// TwinCAT 3 PLC project project
// ProgramVersion: 3.1.4023.0
// libraries:
//   Tc2_Standard, * (Beckhoff Automation GmbH)
//   Tc2_System, * (Beckhoff Automation GmbH)
//   Tc3_Module, * (Beckhoff Automation GmbH)
// project tree:
//   / PlcTask.TcTTO (not stored)
//   POUs/ FB_NAME.TcPOU, I_NAME.TcIO, MAIN.TcPOU, POU.TcPOU, MUL3.TcPOU
// real-time tasks:
//   TASK PlcTask: cycle T#10ms, priority 20, ADS port 350

// ---- POUs/I_NAME.TcIO
INTERFACE I_NAME

PROPERTY Name : STRING
GET
END_GET
SET
END_SET
END_PROPERTY

METHOD NUM : INT
VAR_INPUT
END_VAR
END_METHOD

END_INTERFACE

// ---- POUs/FB_NAME.TcPOU
FUNCTION_BLOCK FB_NAME IMPLEMENTS I_NAME
VAR_INPUT
END_VAR
VAR_OUTPUT
END_VAR
VAR
	m_name : STRING := 'User';
END_VAR

{warning 'add property implementation'}
PROPERTY Name : STRING
GET
Name := m_name;
END_GET
SET
m_name := Name;
END_SET
END_PROPERTY

{warning 'add method implementation '}
METHOD NUM : INT
NUM := LEN(name);
END_METHOD

END_FUNCTION_BLOCK

// ---- POUs/MAIN.TcPOU
PROGRAM MAIN
VAR
END_VAR

POU();

END_PROGRAM

// ---- POUs/POU.TcPOU
PROGRAM POU
VAR
	
	i : INT := 0;
	f : REAL := 0.0;
	elapsed : TIME := TIME#0M0S0MS;
	today : DATE := DATE#2020-01-01;
	message : STRING := '';
	count : BYTE := 0;
	
	A AT %I* : BOOL := FALSE;
	B AT %I* : BOOL := FALSE;
	C AT %I* : BOOL := FALSE;
	D AT %Q* : BOOL := FALSE;
		
	op1 : INT := 1;
	op2 : INT := 2;
	res : REAL := 0.0;
	test : BOOL := FALSE;
	
	tmr1 : TON;
	
	user : I_NAME;
	name : FB_NAME;
	
	
END_VAR

// Single line comment

(* 
	Multiple line comment
*)

// Structured Text statments

i := 0;
f := 0.0;
elapsed := T#1S;
today := D#2020-05-18;
message := 'Good Morning!';

// Operators (strongest to weakest binding)

test := A AND (A AND B); // Brackets have strongest binding

res := MAX(op1,op2); // function

res := EXPT(op1, op2); // Exponentation operator

res := -op1; // Negation operator
B := NOT A; // NOT operator

res := op1 * op2; // Multiplication operator
res := op1 / op2; // Division operator
res := op1 MOD op2; // Modulo operator

res := op1 + op2; // Addition operator
res := op1 - op2; // Subtraction operator

test := op1 < op2; // Less than operator
test := op1 > op2; // Greater than operator
test := op1 <= op2; // Less than or equal to operator
test := op1 >= op2; // Greater than or equal to operator

test := op1 = op2; // Equality operator

C := A AND B; // AND operator

C := A XOR B; // XOR operator

C := A OR B; // OR operator

// IF statement

IF A = B THEN // IF statement
	D := TRUE;
END_IF

IF A = B THEN // IF-ELSE statement
	D := TRUE;
ELSE
	D := FALSE;
END_IF

IF A = B THEN // IF-ELSIF statement
	D := TRUE;
ELSIF A = C THEN
	D := FALSE;
END_IF

// CASE Statement

i := 0;

CASE i OF
	0: A := TRUE;
	1: B := TRUE;
	2: C := TRUE;
ELSE
	D := TRUE;
END_CASE

// FOR statement

f := 0.0;

FOR i := 0 TO 5 BY 1 DO // FOR loop
	f := f + i;
END_FOR

f := 0.0;

FOR i := 0 TO 5 BY 1 DO // FOR loop with EXIT statment
	f := f + i;
	
	IF f > 3 THEN
		EXIT;
	END_IF
END_FOR

// WHILE loop

i := 0;
f := 0.0;

WHILE f < 5 DO // WHILE loop
	i := i + 1;	
	f := f + i;
END_WHILE

i := 0;
f := 0.0;

WHILE f < 5 DO // WHILE loop with EXIT statement
	f := f + i;
	i := i + 1;
	
	IF f > 3 THEN
		EXIT;
	END_IF
END_WHILE

// REPEAT loop

i := 0;
f := 0.0;

REPEAT // REPEAT loop
	f := f + i;
	i := i + 1;
UNTIL f >= 5
END_REPEAT

REPEAT // REPEAT loop with EXIT statment
	f := f + i;
	i := i + 1;
	
	IF f > 3 THEN
		EXIT;
	END_IF
UNTIL f = 5
END_REPEAT

// Timer

D := FALSE;
tmr1(IN := TRUE, PT := T#5S);

IF (tmr1.ET >= T#3S) THEN
	D := TRUE;
END_IF

// Using a function

f := MUL3(1.0, 2.0, 3.0);

// Using an interface

user := name;
user.Name := 'John';
i := user.NUM();

END_PROGRAM

// ---- POUs/MUL3.TcPOU
FUNCTION MUL3 : REAL
VAR_INPUT
	in1 : REAL;
	in2 : REAL;
	in3 : REAL;
END_VAR
VAR
END_VAR

MUL3 := in1 * in2 * in3;

END_FUNCTION
